TYPE ST_SheepingPictureInfo :
STRUCT
	CameraDone	:BOOL;
END_STRUCT
END_TYPE

(* stored: Version 1.1.0.1, ProductVersion 3.1.4024.13
   DUT ST_SheepingPictureInfo: Id {4b056669-1045-469b-861b-b5d29f7f12e0} *)
